TYPE (* DataPanel Modules with medium IO density AI Struct *)
  (* Version 1.0, 2026-01-16, generated *)
  PACKAGE DataPanel::io::MI::AI;
  DataPanel_MI_AI_S : STRUCT
    Pin : USINT := 255;
  END_STRUCT;
END_TYPE
